FUNCTION ArmFK : Points
VAR_INPUT
	theta1:LREAL;
	theta2:LREAL;
END_VAR
VAR
	// 中间变量
	theta1_rad:LREAL;
	theta2_rad:LREAL;
	rr:LREAL;						//r变量被倍福占用了，所以此处用rr
	u:LREAL;
	angle_ACD:LREAL;
	angle_DCE:LREAL;
	angle_ACF:LREAL;
	angle_FCG:LREAL;
	angle_FCI:LREAL;
	
	// 输出
	points : Points;

END_VAR

theta1_rad := DEG_TO_RAD(theta1);
theta2_rad := DEG_TO_RAD(theta2);


rr := SQRT(EXPT((2*w+f*COS(theta1_rad)-g*COS(theta2_rad)),2) + EXPT((f*SIN(theta1_rad)-g*SIN(theta2_rad)),2));  

u := SQRT(EXPT((2*w-g*COS(theta2_rad)),2) + EXPT((-g*SIN(theta2_rad)),2));


angle_ACD := ACOS((rr*rr+f*f-u*u)/(2*rr*f));


angle_DCE := ACOS((rr*rr + i*i -h*h)/(2*rr*i));


angle_ACF := angle_ACD + angle_DCE + DEG_TO_RAD(angle_FCE);


angle_FCG := angle_ACF - theta1_rad;


angle_FCI := PI - angle_FCG;
points.x := w + f*COS(theta1_rad) + n*COS(angle_FCI);
points.y := f*SIN(theta1_rad) + n*SIN(angle_FCI);

ArmFK := points;

END_FUNCTION

(* stored: Version 1.1.0.1, ProductVersion 3.1.4024.13
   POU ArmFK: Id {874f104e-3823-4873-84ee-579597cb6d6e}, SpecialFunc None *)
